// TIA Portal project "LabelerSPM" (V15.1)

(* hardware
DEVICE "S7-1200 station_1"  S7-1200 Station
   slot 0: "Rack_0"  S7-1200 Rack  Rack  V1.0
   slot 1: "PLC_1"  CPU 1212C DC/DC/DC  6ES7 212-1AE40-0XB0  V4.2
*)

// ===== PLC "PLC_1"  CPU 1212C DC/DC/DC =====

VAR_GLOBAL   // PLC tag table "Default tag table"
   "Roll_Pulse" AT %Q0.1 : Bool;
   "Roll_Direction" AT %Q0.3 : Bool;
   "TimeInterrupt" AT %MW0 : Word;
   "DelayBottle" AT %MW2 : Int;
   "SENSORBOTTLE" AT %I0.0 : Bool;
   "SENSORSTAMP" AT %I0.1 : Bool;
   "InterruptBotle" AT %MD4 : Event_Att;
   "RunningBottle" AT %MW8 : Int;
END_VAR

DATA_BLOCK "obj_DB"   // DB1
{ S7_Optimized_Access := 'FALSE' }
VERSION : 0.1
// stored: InstanceOfName obj
"obj"
BEGIN
END_DATA_BLOCK

DATA_BLOCK "Roll"   // DB2, Motion_DB
{ S7_Optimized_Access := 'TRUE' }
AUTHOR : SIMATIC
FAMILY : BasicMC
NAME : TO_PosAx
VERSION : 6.0
// stored: InstanceOfName TO_PositioningAxis
"TO_PositioningAxis"
BEGIN
   // Axis.OnlinePtoModeCU = 16#0000_0002
   // Axis.SelectedChannel2EnumCU = %Q0.3
   // Axis.SelectedChannel1EnumCU = %Q0.1
   // Pulse.MinDeltaDeltaFrequencyCU = 0.004
   // Pulse.MaxDeltaDeltaFrequencyCU = 1.0E+10
   // Pulse.MinDeltaFrequencyCU = 0.005
   // Pulse.MaxDeltaFrequencyCU = 9.5E+9
   // Pulse.MinFrequencyCU = 1.0
   // Pulse.MaxFrequencyCU = 100000.0
   // Pulse.OutputSourceCU = 16#0000_0000
   // Axis.SelectPTO = 1
   // Axis.OnlinePtoIndexCU = 1
   // Axis.LengthUnit.LastDistance = 1010
END_DATA_BLOCK

FUNCTION_BLOCK "obj"   // FB1, SCL
{ S7_Optimized_Access := 'FALSE' }
VERSION : 0.1
   VAR_INPUT
      SignalBottle : Bool;
      SignalLabel : Bool;
      EncoderConv : Bool;
      EncoderRoll : Bool;
      Emerg : Bool;
   END_VAR
   VAR_OUTPUT
      PTOLabel : Bool;
      PTORoll : Bool;
      PTOConv : Bool;
      OutputPrint : Bool;
   END_VAR
   VAR
      config : Bool;
      roundBottle : Bool;
      setPrint : Bool;
      upload : Bool;
      save : Bool;
      "Counter" : Int;
      Pointer : Int;
      control : Struct
         pushConv : Bool;
         pushLabel : Bool;
         runConv : Bool;
         runLabel : Bool;
      END_STRUCT;
      Label : Struct
         Fullstep : Int;
         Microstep : Int;
         Frequency : Real;
         Speed : Real;
         OffsetSpeed : Real;
         Diameter : Real;
         ZeroLength : Real;
         DivLength : Real;
         Ratio : Real;
         Pulses : Real;
         Gear : Real;
      END_STRUCT;
      Conveyor : Struct
         Fullstep : Int;
         Microstep : Int;
         Frequency : Real;
         Speed : Real;
         OffsetSpeed : Real;
         Diameter : Real;
         Ratio : Real;
         Gear : Real;
      END_STRUCT;
      Rolling : Struct
         Fullstep : Int;
         Microstep : Int;
         Frequency : Real;
         Speed : Real;
         OffsetSpeed : Real;
         Diameter : Real;
         Ratio : Real;
         Gear : Real;
      END_STRUCT;
      Bottle : Struct
         Delay : DInt;
         DelayPrint : DInt;
         OffsetLen : Real;
         ExtraLen : Real;
         ZeroLen : Real;   // k/c từ điểm phát hiện đến điểm dán
         ZeroLabel : Real;
         SizeLabel : Real;
         Diameter : Real;
      END_STRUCT;
      stack : Array[0..50] of Struct
         quantity : DInt;
         remning : DInt;
         setAlarm : DInt;
         labSpeed : Real;
         labPosition : Real;
         labLength : Real;
         labLenOff : Real;
      END_STRUCT;
      TimerPrint : TON_TIME;
      DelayPrint : TON_TIME;
   END_VAR
BEGIN
   // #Label.Diameter - mm     #Label.Speed - m/min.       #Label.SizeLabel - mm
   // Freq := (speed*microstep*fullstep)/(time*chuviRulo)  v = 2r*pi*f
   // đo đk chai để xác định tâm chai, tìm điểm dán #Bottle.Diameter / 2

   // Time delay print signal
   IF #SignalLabel THEN
       #setPrint := TRUE;
   END_IF;
   #TimerPrint(IN := #setPrint, PT := #Bottle.DelayPrint);
   #DelayPrint(IN := #TimerPrint.Q, PT := t#200ms);

   IF #TimerPrint.Q THEN
       #OutputPrint := TRUE;
   END_IF;

   IF #DelayPrint.Q THEN
       #OutputPrint := FALSE;
       #setPrint := FALSE;
   END_IF;

   // Labeler position
   #Bottle.Delay := ROUND((60 * (#Bottle.ZeroLen - (#Bottle.Diameter / 2) + #Bottle.OffsetLen)) / #Conveyor.Speed);

   // Conveyor
   #Conveyor.Frequency := ((#Conveyor.Speed + #Conveyor.OffsetSpeed) * #Conveyor.Ratio * 1000) / 60;
   // Rolling - Rolling.speed = 2 * Conveyor.Speed
   #Rolling.Frequency := ((#Rolling.Speed + #Rolling.OffsetSpeed) * #Rolling.Ratio * 1000) / 60;
   // Label Label.speed = Conveyor.Speed
   #Label.Frequency := ((#Label.Speed + #Label.OffsetSpeed) * #Label.Ratio * 1000) / 60;

   // control
   IF #roundBottle THEN
       #Rolling.Speed := 2 * #Conveyor.Speed;
       #Label.Speed := #Conveyor.Speed;
   ELSE
       #Rolling.Speed := #Conveyor.Speed;
       #Label.Speed := #Conveyor.Speed;
   END_IF;

   "RunningBottle" := ATTACH(OB_NR := 40, EVENT := "InterruptBotle", ADD := #SignalBottle);
   #Bottle.OffsetLen := #Bottle.Diameter / 15;
   #Label.Pulses := (#Bottle.ZeroLabel + #Bottle.OffsetLen + #Bottle.ExtraLen) * #Label.Ratio;

   // Config

   IF #config THEN
       #Label.DivLength := TRUNC(#Label.ZeroLength / #Bottle.SizeLabel);
       IF #Label.DivLength < 1 THEN
           #Bottle.ZeroLabel := #Label.ZeroLength;
       ELSE
           #Bottle.ZeroLabel := #Label.ZeroLength - #Label.DivLength * #Bottle.SizeLabel;
       END_IF;

       #Conveyor.Ratio := (#Conveyor.Microstep * #Conveyor.Fullstep * #Conveyor.Gear) / (#Conveyor.Diameter * 3.14159);
       #Rolling.Ratio := (#Rolling.Microstep * #Rolling.Fullstep * #Rolling.Gear) / (#Rolling.Diameter * 3.14159);
       #Label.Ratio := (#Label.Microstep * #Label.Fullstep * #Label.Gear) / (#Label.Diameter * 3.14159);



   END_IF;
END_FUNCTION_BLOCK

FUNCTION_BLOCK "DriveControl"   // FB2, SCL
{ S7_Optimized_Access := 'TRUE' }
VERSION : 0.1
   VAR_INPUT
      Enable_Power : Bool;
      StartMode_Power : Int;
      StopMode_Power : Int;
      Ececute_Relative : Bool;
      Distance_Relative : Real;
      Velocity_Relative : Real;
   END_VAR
   VAR_OUTPUT
      Status_Power : Bool;
      Busy_Power : Bool;
      Error_Power : Bool;
      ErrorID_Power : Word;
      ErrorInfo_Power : Word;
      Done_Relative : Bool;
      Busy_Relative : Bool;
      Command_Relative : Bool;
      Error_Relative : Bool;
      ErrorID_Relative : Word;
      ErrorInfo_Relative : Word;
   END_VAR
   VAR_IN_OUT
      Axis : TO_Axis;
      Axis_Position : TO_PositioningAxis;
   END_VAR
   VAR
      MC_Power : MC_Power;
      MC_MoveRelative : MC_MoveRelative;
   END_VAR
BEGIN


   #MC_Power(Axis := #Axis,
             Enable := #Enable_Power,
             StartMode := #StartMode_Power,
             StopMode := #StopMode_Power,
             Status => #Status_Power,
             Busy => #Busy_Power,
             Error => #Error_Power,
             ErrorID => #ErrorID_Power,
             ErrorInfo => #ErrorInfo_Power);

   #MC_MoveRelative(Axis := #Axis_Position,
                    Execute := #Ececute_Relative,
                    Distance := #Distance_Relative,
                    Velocity := #Velocity_Relative,
                    Done => #Done_Relative,
                    Busy => #Busy_Relative,
                    CommandAborted => #Command_Relative,
                    Error => #Error_Relative,
                    ErrorID => #ErrorID_Relative,
                    ErrorInfo => #ErrorInfo_Relative);
END_FUNCTION_BLOCK

FUNCTION "ConvertI/O" : Void   // FC1, SCL
{ S7_Optimized_Access := 'TRUE' }
VERSION : 0.1
BEGIN
END_FUNCTION

ORGANIZATION_BLOCK "Main"   // OB1, LAD, ProgramCycle
TITLE = "Main Program Sweep (Cycle)"
{ S7_Optimized_Access := 'TRUE' }
VERSION : 0.1
   VAR_INPUT
      Initial_Call : Bool;   // Initial call of this OB
      Remanence : Bool;   // =True, if remanent data are available
   END_VAR
BEGIN

REGION Network 1
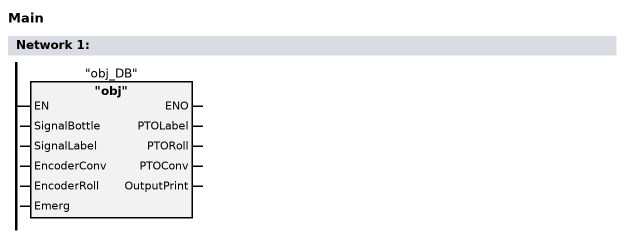
   RUNG wire#powerrail
      "obj_DB"(SignalBottle :=, SignalLabel :=, EncoderConv :=, EncoderRoll :=, Emerg :=, PTOLabel =>, PTORoll =>, PTOConv =>, OutputPrint =>)
   END_RUNG
   // the same network as SCL:
   "obj_DB"();   // "obj"
END_REGION
END_ORGANIZATION_BLOCK

ORGANIZATION_BLOCK "Delay labeler"   // OB20, SCL, TimeDelayInterrupt
{ S7_Optimized_Access := 'TRUE' }
VERSION : 0.1
   VAR_INPUT
      Sign : Word;   // Identifier input (SIGN) passed to triggering call of SRT_DINT
   END_VAR
BEGIN
   "obj_DB".control.runLabel := TRUE;
END_ORGANIZATION_BLOCK

ORGANIZATION_BLOCK "Cyclic Control"   // OB30, SCL, CyclicInterrupt
{ S7_Optimized_Access := 'TRUE' }
VERSION : 0.1
   VAR_INPUT
      Initial_Call : Bool;   // Initial call of this OB
      Event_Count : Int;   // Events discarded
   END_VAR
BEGIN
END_ORGANIZATION_BLOCK

ORGANIZATION_BLOCK "Find_Bottle"   // OB40, SCL, HWProcessInterrupt
{ S7_Optimized_Access := 'TRUE' }
VERSION : 0.1
   VAR_INPUT
      LADDR : Hw_Io;   // Hardware identifier
      USI : Word;   // User structure identifier
      IChannel : USInt;   // Interrupt channel number
      EventType : Byte;   // EventType
   END_VAR
BEGIN
   "DelayBottle" := SRT_DINT(OB_NR := 20, DTIME := "obj_DB".Bottle.Delay, SIGN := "TimeInterrupt");
END_ORGANIZATION_BLOCK

ORGANIZATION_BLOCK "Find_Stamp"   // OB41, SCL, HWProcessInterrupt
{ S7_Optimized_Access := 'TRUE' }
VERSION : 0.1
   VAR_INPUT
      LADDR : Hw_Io;   // Hardware identifier
      USI : Word;   // User structure identifier
      IChannel : USInt;   // Interrupt channel number
      EventType : Byte;   // EventType
   END_VAR
BEGIN
END_ORGANIZATION_BLOCK